{attribute addProperty BoxType "EL2032--0000"}
{attribute addProperty Id "DiagAT %I*BOOL81"}
{attribute addProperty CRC "1289020322"}
{attribute addProperty SizeInBites "8"}
{attribute addProperty SizeInBytes "1"}
TYPE Diag_4CD4E3A2 :
STRUCT
	{attribute addProperty Name "Diag"}
	Diag AT %I* : BOOL;
END_STRUCT
END_TYPE

(* stored: Version 1.2.0.0, ProductVersion 3.1.4024.9
   DUT Diag_4CD4E3A2: Id {232ab21b-5176-48df-9a7f-151fb5b81465} *)
